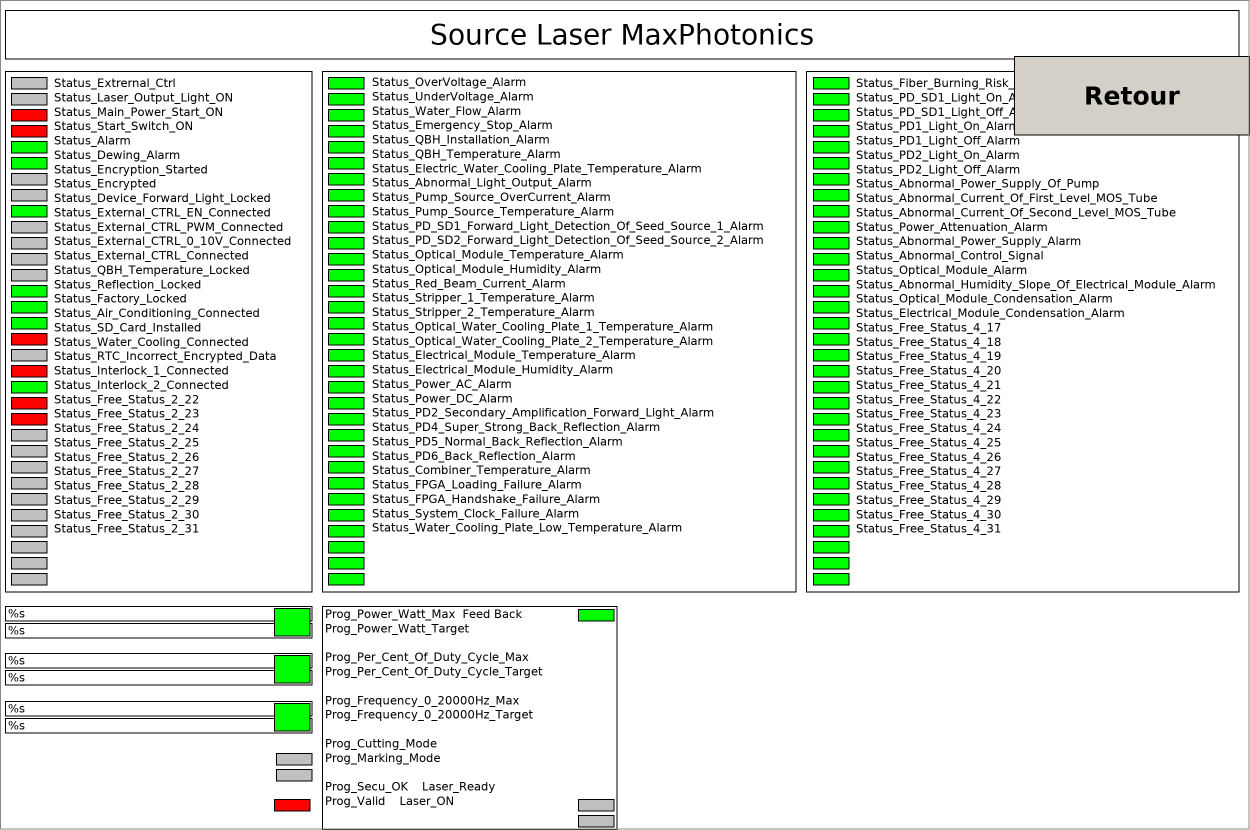
VISUALIZATION Laser_Source_1  // 1250x830
VAR_IN_OUT
	prog_secu_ok	:BOOL;
END_VAR
    Rectangle (806,71 433x521)
    Rectangle (322,71 474x521)
    Rectangle (5,71 307x521)
    Rectangle (51,75 256x516), "Status_Extrernal_Ctrl Status_Laser_Output_Light_ON Status_Main_Power_Start_ON Status_Start_Switch_ON Status_Alarm Status_Dewing_Alarm Status_Encryption_Started Status_Encrypted Status_Device_Forward_Light_Locked Status_External_CTRL_EN_Connected Status_External_CTRL_PWM_Connected Status_External_CTRL_0_10V_Connected Status_External_CTRL_Connected Status_QBH_Temperature_Locked Status_Reflection_Locked Status_Factory_Locked Status_Air_Conditioning_Connected Status_SD_Card_Installed Status_Water_Cooling_Connected Status_RTC_Incorrect_Encrypted_Data Status_Interlock_1_Connected Status_Interlock_2_Connected Status_Free_Status_2_22 Status_Free_Status_2_23 Status_Free_Status_2_24 Status_Free_Status_2_25 Status_Free_Status_2_26 Status_Free_Status_2_27 Status_Free_Status_2_28 Status_Free_Status_2_29 Status_Free_Status_2_30 Status_Free_Status_2_31"
    Rectangle (369,74 424x515), "Status_OverVoltage_Alarm Status_UnderVoltage_Alarm Status_Water_Flow_Alarm Status_Emergency_Stop_Alarm Status_QBH_Installation_Alarm Status_QBH_Temperature_Alarm Status_Electric_Water_Cooling_Plate_Temperature_Alarm Status_Abnormal_Light_Output_Alarm Status_Pump_Source_OverCurrent_Alarm Status_Pump_Source_Temperature_Alarm Status_PD_SD1_Forward_Light_Detection_Of_Seed_Source_1_Alarm Status_PD_SD2_Forward_Light_Detection_Of_Seed_Source_2_Alarm Status_Optical_Module_Temperature_Alarm Status_Optical_Module_Humidity_Alarm Status_Red_Beam_Current_Alarm Status_Stripper_1_Temperature_Alarm Status_Stripper_2_Temperature_Alarm Status_Optical_Water_Cooling_Plate_1_Temperature_Alarm Status_Optical_Water_Cooling_Plate_2_Temperature_Alarm Status_Electrical_Module_Temperature_Alarm Status_Electrical_Module_Humidity_Alarm Status_Power_AC_Alarm Status_Power_DC_Alarm Status_PD2_Secondary_Amplification_Forward_Light_Alarm Status_PD4_Super_Strong_Back_Reflection_Alarm Status_PD5_Normal_Back_Reflection_Alarm Status_PD6_Back_Reflection_Alarm Status_Combiner_Temperature_Alarm Status_FPGA_Loading_Failure_Alarm Status_FPGA_Handshake_Failure_Alarm Status_System_Clock_Failure_Alarm Status_Water_Cooling_Plate_Low_Temperature_Alarm"
    Rectangle (11,77 36x12), colour toggle: IO_SOURCE_MAXPHOTONICS.STATUS_2.0
    Rectangle (11,93 36x12), colour toggle: IO_SOURCE_MAXPHOTONICS.STATUS_2.1
    Rectangle (11,109 36x12), colour toggle: IO_SOURCE_MAXPHOTONICS.STATUS_2.2
    Rectangle (11,125 36x12), colour toggle: IO_SOURCE_MAXPHOTONICS.STATUS_2.3
    Rectangle (328,77 36x12), colour toggle: IO_SOURCE_MAXPHOTONICS.STATUS_3.0
    Rectangle (328,93 36x12), colour toggle: IO_SOURCE_MAXPHOTONICS.STATUS_3.1
    Rectangle (328,109 36x12), colour toggle: IO_SOURCE_MAXPHOTONICS.STATUS_3.2
    Rectangle (328,125 36x12), colour toggle: IO_SOURCE_MAXPHOTONICS.STATUS_3.3
    Rectangle (328,141 36x12), colour toggle: IO_SOURCE_MAXPHOTONICS.STATUS_3.4
    Rectangle (328,157 36x12), colour toggle: IO_SOURCE_MAXPHOTONICS.STATUS_3.5
    Rectangle (328,173 36x12), colour toggle: IO_SOURCE_MAXPHOTONICS.STATUS_3.6
    Rectangle (328,189 36x12), colour toggle: IO_SOURCE_MAXPHOTONICS.STATUS_3.7
    Rectangle (328,205 36x12), colour toggle: IO_SOURCE_MAXPHOTONICS.STATUS_3.8
    Rectangle (328,221 36x12), colour toggle: IO_SOURCE_MAXPHOTONICS.STATUS_3.9
    Rectangle (328,237 36x12), colour toggle: IO_SOURCE_MAXPHOTONICS.STATUS_3.10
    Rectangle (328,253 36x12), colour toggle: IO_SOURCE_MAXPHOTONICS.STATUS_3.11
    Rectangle (328,269 36x12), colour toggle: IO_SOURCE_MAXPHOTONICS.STATUS_3.12
    Rectangle (328,285 36x12), colour toggle: IO_SOURCE_MAXPHOTONICS.STATUS_3.13
    Rectangle (328,301 36x12), colour toggle: IO_SOURCE_MAXPHOTONICS.STATUS_3.14
    Rectangle (328,317 36x12), colour toggle: IO_SOURCE_MAXPHOTONICS.STATUS_3.15
    Rectangle (328,333 36x12), colour toggle: IO_SOURCE_MAXPHOTONICS.STATUS_3.16
    Rectangle (328,349 36x12), colour toggle: IO_SOURCE_MAXPHOTONICS.STATUS_3.17
    Rectangle (328,365 36x12), colour toggle: IO_SOURCE_MAXPHOTONICS.STATUS_3.18
    Rectangle (328,381 36x12), colour toggle: IO_SOURCE_MAXPHOTONICS.STATUS_3.19
    Rectangle (328,397 36x12), colour toggle: IO_SOURCE_MAXPHOTONICS.STATUS_3.20
    Rectangle (328,413 36x12), colour toggle: IO_SOURCE_MAXPHOTONICS.STATUS_3.21
    Rectangle (328,429 36x12), colour toggle: IO_SOURCE_MAXPHOTONICS.STATUS_3.22
    Rectangle (328,445 36x12), colour toggle: IO_SOURCE_MAXPHOTONICS.STATUS_3.23
    Rectangle (328,461 36x12), colour toggle: IO_SOURCE_MAXPHOTONICS.STATUS_3.24
    Rectangle (328,477 36x12), colour toggle: IO_SOURCE_MAXPHOTONICS.STATUS_3.25
    Rectangle (328,493 36x12), colour toggle: IO_SOURCE_MAXPHOTONICS.STATUS_3.26
    Rectangle (328,509 36x12), colour toggle: IO_SOURCE_MAXPHOTONICS.STATUS_3.27
    Rectangle (328,525 36x12), colour toggle: IO_SOURCE_MAXPHOTONICS.STATUS_3.28
    Rectangle (328,541 36x12), colour toggle: IO_SOURCE_MAXPHOTONICS.STATUS_3.29
    Rectangle (328,557 36x12), colour toggle: IO_SOURCE_MAXPHOTONICS.STATUS_3.30
    Rectangle (328,573 36x12), colour toggle: IO_SOURCE_MAXPHOTONICS.STATUS_3.31
    Rectangle (11,141 36x12), colour toggle: IO_SOURCE_MAXPHOTONICS.STATUS_2.4
    Rectangle (11,157 36x12), colour toggle: IO_SOURCE_MAXPHOTONICS.STATUS_2.5
    Rectangle (11,173 36x12), colour toggle: IO_SOURCE_MAXPHOTONICS.STATUS_2.6
    Rectangle (11,189 36x12), colour toggle: IO_SOURCE_MAXPHOTONICS.STATUS_2.7
    Rectangle (11,205 36x12), colour toggle: IO_SOURCE_MAXPHOTONICS.STATUS_2.8
    Rectangle (11,221 36x12), colour toggle: IO_SOURCE_MAXPHOTONICS.STATUS_2.9
    Rectangle (11,237 36x12), colour toggle: IO_SOURCE_MAXPHOTONICS.STATUS_2.10
    Rectangle (11,253 36x12), colour toggle: IO_SOURCE_MAXPHOTONICS.STATUS_2.11
    Rectangle (11,269 36x12), colour toggle: IO_SOURCE_MAXPHOTONICS.STATUS_2.12
    Rectangle (11,285 36x12), colour toggle: IO_SOURCE_MAXPHOTONICS.STATUS_2.13
    Rectangle (11,301 36x12), colour toggle: IO_SOURCE_MAXPHOTONICS.STATUS_2.14
    Rectangle (11,317 36x12), colour toggle: IO_SOURCE_MAXPHOTONICS.STATUS_2.15
    Rectangle (11,333 36x12), colour toggle: IO_SOURCE_MAXPHOTONICS.STATUS_2.16
    Rectangle (11,349 36x12), colour toggle: IO_SOURCE_MAXPHOTONICS.STATUS_2.17
    Rectangle (11,365 36x12), colour toggle: IO_SOURCE_MAXPHOTONICS.STATUS_2.18
    Rectangle (11,381 36x12), colour toggle: IO_SOURCE_MAXPHOTONICS.STATUS_2.19
    Rectangle (11,397 36x12), colour toggle: IO_SOURCE_MAXPHOTONICS.STATUS_2.20
    Rectangle (11,413 36x12), colour toggle: IO_SOURCE_MAXPHOTONICS.STATUS_2.21
    Rectangle (11,429 36x12), colour toggle: IO_SOURCE_MAXPHOTONICS.STATUS_2.22
    Rectangle (11,445 36x12), colour toggle: IO_SOURCE_MAXPHOTONICS.STATUS_2.23
    Rectangle (11,461 36x12), colour toggle: IO_SOURCE_MAXPHOTONICS.STATUS_2.24
    Rectangle (11,477 36x12), colour toggle: IO_SOURCE_MAXPHOTONICS.STATUS_2.25
    Rectangle (11,493 36x12), colour toggle: IO_SOURCE_MAXPHOTONICS.STATUS_2.26
    Rectangle (11,509 36x12), colour toggle: IO_SOURCE_MAXPHOTONICS.STATUS_2.27
    Rectangle (11,525 36x12), colour toggle: IO_SOURCE_MAXPHOTONICS.STATUS_2.28
    Rectangle (11,541 36x12), colour toggle: IO_SOURCE_MAXPHOTONICS.STATUS_2.29
    Rectangle (11,557 36x12), colour toggle: IO_SOURCE_MAXPHOTONICS.STATUS_2.30
    Rectangle (11,573 36x12), colour toggle: IO_SOURCE_MAXPHOTONICS.STATUS_2.31
    Rectangle (853,75 384x513), "Status_Fiber_Burning_Risk_Alarm Status_PD_SD1_Light_On_Alarm Status_PD_SD1_Light_Off_Alarm Status_PD1_Light_On_Alarm Status_PD1_Light_Off_Alarm Status_PD2_Light_On_Alarm Status_PD2_Light_Off_Alarm Status_Abnormal_Power_Supply_Of_Pump Status_Abnormal_Current_Of_First_Level_MOS_Tube Status_Abnormal_Current_Of_Second_Level_MOS_Tube Status_Power_Attenuation_Alarm Status_Abnormal_Power_Supply_Alarm Status_Abnormal_Control_Signal Status_Optical_Module_Alarm Status_Abnormal_Humidity_Slope_Of_Electrical_Module_Alarm Status_Optical_Module_Condensation_Alarm Status_Electrical_Module_Condensation_Alarm Status_Free_Status_4_17 Status_Free_Status_4_18 Status_Free_Status_4_19 Status_Free_Status_4_20 Status_Free_Status_4_21 Status_Free_Status_4_22 Status_Free_Status_4_23 Status_Free_Status_4_24 Status_Free_Status_4_25 Status_Free_Status_4_26 Status_Free_Status_4_27 Status_Free_Status_4_28 Status_Free_Status_4_29 Status_Free_Status_4_30 Status_Free_Status_4_31"
    Rectangle (813,77 36x12), colour toggle: IO_SOURCE_MAXPHOTONICS.STATUS_4.0
    Rectangle (813,93 36x12), colour toggle: IO_SOURCE_MAXPHOTONICS.STATUS_4.1
    Rectangle (813,109 36x12), colour toggle: IO_SOURCE_MAXPHOTONICS.STATUS_4.2
    Rectangle (813,125 36x12), colour toggle: IO_SOURCE_MAXPHOTONICS.STATUS_4.3
    Rectangle (813,141 36x12), colour toggle: IO_SOURCE_MAXPHOTONICS.STATUS_4.4
    Rectangle (813,157 36x12), colour toggle: IO_SOURCE_MAXPHOTONICS.STATUS_4.5
    Rectangle (813,173 36x12), colour toggle: IO_SOURCE_MAXPHOTONICS.STATUS_4.6
    Rectangle (813,189 36x12), colour toggle: IO_SOURCE_MAXPHOTONICS.STATUS_4.7
    Rectangle (813,205 36x12), colour toggle: IO_SOURCE_MAXPHOTONICS.STATUS_4.8
    Rectangle (813,221 36x12), colour toggle: IO_SOURCE_MAXPHOTONICS.STATUS_4.9
    Rectangle (813,237 36x12), colour toggle: IO_SOURCE_MAXPHOTONICS.STATUS_4.10
    Rectangle (813,253 36x12), colour toggle: IO_SOURCE_MAXPHOTONICS.STATUS_4.11
    Rectangle (813,269 36x12), colour toggle: IO_SOURCE_MAXPHOTONICS.STATUS_4.12
    Rectangle (813,285 36x12), colour toggle: IO_SOURCE_MAXPHOTONICS.STATUS_4.13
    Rectangle (813,301 36x12), colour toggle: IO_SOURCE_MAXPHOTONICS.STATUS_4.14
    Rectangle (813,317 36x12), colour toggle: IO_SOURCE_MAXPHOTONICS.STATUS_4.15
    Rectangle (813,333 36x12), colour toggle: IO_SOURCE_MAXPHOTONICS.STATUS_4.16
    Rectangle (813,349 36x12), colour toggle: IO_SOURCE_MAXPHOTONICS.STATUS_4.17
    Rectangle (813,365 36x12), colour toggle: IO_SOURCE_MAXPHOTONICS.STATUS_4.18
    Rectangle (813,381 36x12), colour toggle: IO_SOURCE_MAXPHOTONICS.STATUS_4.19
    Rectangle (813,397 36x12), colour toggle: IO_SOURCE_MAXPHOTONICS.STATUS_4.20
    Rectangle (813,413 36x12), colour toggle: IO_SOURCE_MAXPHOTONICS.STATUS_4.21
    Rectangle (813,429 36x12), colour toggle: IO_SOURCE_MAXPHOTONICS.STATUS_4.22
    Rectangle (813,445 36x12), colour toggle: IO_SOURCE_MAXPHOTONICS.STATUS_4.23
    Rectangle (813,461 36x12), colour toggle: IO_SOURCE_MAXPHOTONICS.STATUS_4.24
    Rectangle (813,477 36x12), colour toggle: IO_SOURCE_MAXPHOTONICS.STATUS_4.25
    Rectangle (813,493 36x12), colour toggle: IO_SOURCE_MAXPHOTONICS.STATUS_4.26
    Rectangle (813,509 36x12), colour toggle: IO_SOURCE_MAXPHOTONICS.STATUS_4.27
    Rectangle (813,525 36x12), colour toggle: IO_SOURCE_MAXPHOTONICS.STATUS_4.28
    Rectangle (813,541 36x12), colour toggle: IO_SOURCE_MAXPHOTONICS.STATUS_4.29
    Rectangle (813,557 36x12), colour toggle: IO_SOURCE_MAXPHOTONICS.STATUS_4.30
    Rectangle (813,573 36x12), colour toggle: IO_SOURCE_MAXPHOTONICS.STATUS_4.31
    Rectangle (5,10 1234x49), "Source Laser MaxPhotonics"
    Rectangle (5,606 307x15), "%s", text variable: IO_SOURCE_MAXPHOTONICS.PLC_Prog_Power_Watt_Max
    Rectangle (322,606 295x224), "Prog_Power_Watt_Max Feed Back Prog_Power_Watt_Target Prog_Per_Cent_Of_Duty_Cycle_Max Prog_Per_Cent_Of_Duty_Cycle_Target Prog_Frequency_0_20000Hz_Max Prog_Frequency_0_20000Hz_Target Prog_Cutting_Mode Prog_Marking_Mode Prog_Secu_OK Laser_Ready Prog_Valid Laser_ON"
    Rectangle (5,623 307x15), "%s", text variable: IO_SOURCE_MAXPHOTONICS.PLC_Prog_Power_Watt_Target
    Rectangle (5,653 307x15), "%s", text variable: IO_SOURCE_MAXPHOTONICS.Prog_Per_Cent_Of_Duty_Cycle_Max
    Rectangle (5,670 307x15), "%s", text variable: IO_SOURCE_MAXPHOTONICS.Prog_Per_Cent_Of_Duty_Cycle_Target
    Rectangle (5,701 307x15), "%s", text variable: IO_SOURCE_MAXPHOTONICS.Prog_Frequency_0_20000Hz_Max
    Rectangle (5,718 307x15), "%s", text variable: IO_SOURCE_MAXPHOTONICS.Prog_Frequency_0_20000Hz_Target
    Rectangle (276,753 36x12), colour toggle: IO_SOURCE_MAXPHOTONICS.Prog_Cutting_Mode
    Rectangle (276,769 36x12), colour toggle: IO_SOURCE_MAXPHOTONICS.Prog_Marking_Mode
    Rectangle (274,799 36x12), colour toggle: (Prog_Secu_OK)
    Rectangle (274,608 36x28), colour toggle: IO_SOURCE_MAXPHOTONICS.Prog_Defaut_power_Watt_Target
    Rectangle (274,655 36x28), colour toggle: IO_SOURCE_MAXPHOTONICS.Prog_Defaut_Per_Cent_Of_Duty_Cycle_Target
    Rectangle (274,703 36x28), colour toggle: IO_SOURCE_MAXPHOTONICS.Prog_Defaut_Laser_Frequency_Of_PWM_Wave_Target
    Rectangle (578,609 36x12), colour toggle: IO_SOURCE_MAXPHOTONICS.Prog_Defaut_Perc_Cent_Of_Laser_Output_Power_FeedBack
    Rectangle (578,815 36x12), colour toggle: IO_SOURCE_MAXPHOTONICS.STATUS_2.1
    Rectangle (578,799 36x12), colour toggle: IO_SOURCE_MAXPHOTONICS.STATUS_2.1
    Rectangle (1014,56 236x79), "Retour"
        OnMouseClick: change screen: MenuPrincipal
END_VISUALIZATION

(* stored: Version 1.1.0.1
   Visu Laser_Source_1: Id {993c9eaa-0b2f-4ea7-b4bc-8907b38e7a6a} *)
